INTERFACE I_WStringBuilder

METHOD PUBLIC Append : I_WStringBuilder // Append text to the current build string.
VAR_INPUT
	text : WSTRING; // Text to append to current build string
END_VAR
END_METHOD

METHOD PUBLIC AppendAny : I_WStringBuilder // Append text to the current build string.
VAR_INPUT
	value : ANY; // Value to append to current build string
END_VAR
END_METHOD

METHOD PUBLIC Clear : I_WStringBuilder // Clear the current build string.
VAR_INPUT
END_VAR
END_METHOD

METHOD PUBLIC Insert : I_WStringBuilder
VAR_INPUT
	text	 : WSTRING;	// Text to append to current build string
	position : INT;		// Insert position (Index)
END_VAR
END_METHOD

METHOD PUBLIC Reset : I_WStringBuilder //Reset current build string to an empty string.
VAR_INPUT
END_VAR
END_METHOD

METHOD PUBLIC Set : I_WStringBuilder
VAR_INPUT
	text : WSTRING; //Text to append to current build string
END_VAR
END_METHOD

METHOD PUBLIC ToString : T_MaxString // Returns current build string.
END_METHOD

METHOD PUBLIC ToWString : WSTRING // Returns current build string.
VAR_INPUT
END_VAR
END_METHOD

END_INTERFACE

(* stored: Version 1.1.0.1
   Itf I_WStringBuilder: Id {0f839401-1630-4a3e-a354-b4183d910e4d}
   Method Append: Id {5b84f2fa-9eec-4818-bf9a-f51c532cd7a8}
   Method AppendAny: Id {50962844-dc96-48a9-b96c-61ff3cc1c883}
   Method Clear: Id {903947cc-da45-4cd9-af83-c56af290984c}
   Method Insert: Id {94c543e0-a320-4fb2-9549-d1d34717fad1}
   Method Reset: Id {20e30e21-ada1-4315-84a6-d144832187ac}
   Method Set: Id {2e011a06-200f-43a2-a244-031e632cb2af}
   Method ToString: Id {efa1d400-49a7-4909-be91-503ebc03e687}
   Method ToWString: Id {f9a5695d-b4a1-46ef-8fbd-162f35afc064} *)
